FUNCTION_BLOCK DIChannel IMPLEMENTS I_DigitalInput
VAR
	input AT %I* : BOOL;
END_VAR

PROPERTY PUBLIC bState : BOOL
GET
bState := input;
END_GET
END_PROPERTY

END_FUNCTION_BLOCK

(* stored: Version 1.1.0.1, ProductVersion 3.1.4024.6
   POU DIChannel: Id {cf59d0d9-9926-4c93-8169-8f9a140478e6}, SpecialFunc None
   Property bState: Id {e7b38e79-1425-4a3b-a0f4-1203945e399b}
   Get Get: Id {ad2e312a-5057-43f5-997a-c2b808464078} *)
